// TwinCAT 3 PLC project Plc
// ProgramVersion: 3.1.4023.0
// libraries:
//   Tc2_Standard, * (Beckhoff Automation GmbH)
//   Tc2_System, * (Beckhoff Automation GmbH)
//   Tc2_Utilities, * (Beckhoff Automation GmbH)
//   Tc3_Module, * (Beckhoff Automation GmbH)
// project tree:
//   LinkedList/Master/ FB_LinkedList_Master.TcPOU, ITF_LinkedList_Master.TcIO
//   LinkedList/Node/ FB_LinkedList_Node.TcPOU, ITF_LinkedList_Node.TcIO
//   / PlcTask.TcTTO
//   POUs/Cars/ FB_Car.TcPOU, FB_CarGroup.TcPOU, ITF_Car.TcIO
//   POUs/ MAIN.TcPOU, PERFORMANCE.TcPOU
// real-time tasks:
//   TASK PlcTask: cycle T#10ms, priority 20, ADS port 350

CONFIGURATION Plc
    RESOURCE PLC ON TwinCAT3
        TASK PlcTask(INTERVAL := T#10ms, PRIORITY := 20);
        PROGRAM MAIN WITH PlcTask : MAIN;
        PROGRAM PERFORMANCE WITH PlcTask : PERFORMANCE;
    END_RESOURCE
END_CONFIGURATION

// ---- LinkedList/Master/ITF_LinkedList_Master.TcIO
INTERFACE ITF_LinkedList_Master EXTENDS ITF_LinkedList_Node

METHOD mListAdd : BOOL
VAR_INPUT
	itfNode:	ITF_LinkedList_Node;
END_VAR
END_METHOD

METHOD mListRemove : BOOL
VAR_INPUT
	itfNode:	ITF_LinkedList_Node;
END_VAR
END_METHOD

END_INTERFACE

// ---- LinkedList/Node/ITF_LinkedList_Node.TcIO
INTERFACE ITF_LinkedList_Node EXTENDS __SYSTEM.IQueryInterface

PROPERTY p_IsLinkMaster : BOOL
GET
END_GET
END_PROPERTY

PROPERTY p_ListNext : ITF_LinkedList_Node
GET
END_GET
SET
END_SET
END_PROPERTY

PROPERTY p_ListPrevious : ITF_LinkedList_Node
GET
END_GET
SET
END_SET
END_PROPERTY

END_INTERFACE

// ---- POUs/Cars/ITF_Car.TcIO
INTERFACE ITF_Car

PROPERTY p_Locked : BOOL
GET
END_GET
SET
END_SET
END_PROPERTY

END_INTERFACE

// ---- POUs/MAIN.TcPOU
PROGRAM MAIN
VAR
	fbCarFleet:		FB_CarGroup;
	fbCar_Red:		FB_Car;
	fbCar_Green:	FB_Car;
	fbCar_Blue:		FB_Car;

	fbGarage:		FB_CarGroup;
	fbCorvette:		FB_Car := ( p_LinkMaster := fbGarage );
	fbMustang:		FB_Car := ( p_LinkMaster := fbGarage );

	//Triggers
	xSellCar:		BOOL;
	xBuyCar:		BOOL;
END_VAR

VAR_TEMP
	{attribute 'hide'} 
	pCar:			POINTER TO FB_Car;
END_VAR


IF xSellCar THEN
	xSellCar := FALSE; //Reset trigger
	//Get last car in the garage list and sell it to the fleet
	IF __QUERYPOINTER(fbGarage.mListGetNode( fbGarage.ListLength - 1), pCar) THEN
		pCar^.p_LinkMaster := fbCarFleet;
	END_IF
END_IF

IF xBuyCar THEN
	xBuyCar := FALSE; //Reset trigger
	//Get first car from the fleed and add it to the garage
	IF __QUERYPOINTER(fbCarFleet.mListGetNode(0), pCar) THEN
		pCar^.p_LinkMaster := fbGarage;
	END_IF
END_IF

END_PROGRAM

// ---- POUs/Cars/FB_CarGroup.TcPOU
FUNCTION_BLOCK FB_CarGroup EXTENDS FB_LinkedList_Master IMPLEMENTS ITF_Car
VAR_INPUT
END_VAR
VAR_OUTPUT
END_VAR
VAR
END_VAR

{attribute 'monitoring' := 'call'}
PROPERTY p_Locked : BOOL
GET
VAR
	i:		UINT;
	itfCar:	ITF_Car;
END_VAR
p_Locked := TRUE;

FOR i := 0 TO ListLength DO
	IF __QUERYINTERFACE( mListGetNode(i), itfCar) THEN
		p_Locked R= NOT itfCar.p_Locked;
	END_IF
END_FOR
END_GET
SET
VAR
	i:		UINT;
	itfCar:	ITF_Car;
END_VAR
FOR i := 0 TO ListLength DO
	IF __QUERYINTERFACE( mListGetNode(i), itfCar) THEN
		itfCar.p_Locked := p_Locked;
	END_IF
END_FOR
END_SET
END_PROPERTY

END_FUNCTION_BLOCK

// ---- LinkedList/Master/FB_LinkedList_Master.TcPOU
{attribute 'hide_all_locals'}
FUNCTION_BLOCK FB_LinkedList_Master IMPLEMENTS ITF_LinkedList_Master

VAR_OUTPUT
	ListLength:		UINT;	//Length of the linked list
END_VAR

VAR
	itfHead:	ITF_LinkedList_Node;
	itfTail:	ITF_LinkedList_Node;
	
	{attribute 'no_copy'}
	it:			UINT; 					//Local iterator
	{attribute 'no_copy'}
	itfIt:		ITF_LinkedList_Node;	//Iterated node
END_VAR

METHOD mListAdd : BOOL
VAR_INPUT
	itfNode:	ITF_LinkedList_Node;
END_VAR
IF itfNode <> 0 THEN
	IF ListLength = 0 THEN
		//--Empty list--
		itfHead 				:= itfNode;
		itfTail 				:= itfNode;
		itfNode.p_ListPrevious 	:= THIS^;
		itfNode.p_ListNext		:= THIS^;
	ELSE
		//--Existing list--
		itfTail.p_ListNext 		:= itfNode;
		itfNode.p_ListNext		:= THIS^;
		itfNode.p_ListPrevious	:= itfTail;
		itfTail					:= itfNode;
	END_IF
	
	ListLength := ListLength + 1;
END_IF
END_METHOD

METHOD mListGetNode : ITF_LinkedList_Node
VAR_INPUT
	i:		UINT; //0 => Length - 1
END_VAR
//Reread/init
IF it = 0 THEN
	itfIt  	:= itfHead;
END_IF

//Reset to head
IF i = 0 THEN
	itfIt 	:= itfHead;
	it		:= 0;	
END_IF

WHILE it < i AND_THEN itfIt <> 0 AND_THEN NOT itfIt.p_IsLinkMaster  DO
	itfIt	:= itfIt.p_ListNext;
	it		:= it + 1; 
END_WHILE

WHILE it > i AND_THEN itfIt <> 0 AND_THEN NOT itfIt.p_IsLinkMaster DO
	itfIt	:= itfIt.p_ListPrevious;
	it		:= it - 1;
END_WHILE

IF itfIt <> 0 AND_THEN NOT itfIt.p_IsLinkMaster THEN
	//Node found, return interface
	mListGetNode := itfIt;
ELSE
	//Something went wrong, reset to head
	itfIt 	:= itfHead;
	it		:= 0;
END_IF
END_METHOD

METHOD mListRemove : BOOL
VAR_INPUT
	itfNode:	ITF_LinkedList_Node;
END_VAR
//Improve: Check if node is indeed in the list of this master

IF itfNode <> 0 THEN
	
	IF itfNode.p_ListPrevious <> 0 THEN
		
		IF itfNode.p_ListNext <> 0 THEN
			itfNode.p_ListPrevious.p_ListNext := itfNode.p_ListNext;
			itfNode.p_ListNext.p_ListPrevious := itfNode.p_ListPrevious;
		ELSE
			itfNode.p_ListPrevious.p_ListNext := 0;
		END_IF
		
		mListRemove := TRUE;
	END_IF

	itfNode.p_ListNext 		:= 0;
	itfNode.p_ListPrevious	:= 0;
END_IF

IF mListRemove THEN
	ListLength := MAX(0,ListLength - 1);
	
	//Reset iterator to beginning we don't know where the nodes is removed and recounting is needed
	it		:= 0;
	itfIt	:= itfHead;
END_IF
END_METHOD

PROPERTY p_IsLinkMaster : BOOL
GET
p_IsLinkMaster := TRUE;
END_GET
END_PROPERTY

PROPERTY p_ListNext : ITF_LinkedList_Node
GET
p_ListNext := itfHead;
END_GET
SET
itfHead := p_ListNext;
END_SET
END_PROPERTY

PROPERTY p_ListPrevious : ITF_LinkedList_Node
GET
p_ListPrevious := itfTail;
END_GET
SET
itfTail := p_ListPrevious;
END_SET
END_PROPERTY

END_FUNCTION_BLOCK

// ---- POUs/Cars/FB_Car.TcPOU
{attribute 'hide_all_locals'}
FUNCTION_BLOCK FB_Car EXTENDS FB_LinkedList_Node IMPLEMENTS ITF_Car

VAR
	Locked:		BOOL;
END_VAR

METHOD FB_init : BOOL
VAR_INPUT
	bInitRetains : 	BOOL; // if TRUE, the retain variables are initialized (warm start / cold start)
	bInCopyCode : 	BOOL;  // if TRUE, the instance afterwards gets moved into the copy code (online change)
END_VAR
p_LinkMaster := MAIN.fbCarFleet;
END_METHOD

{attribute 'monitoring' := 'call'}
PROPERTY p_Locked : BOOL
GET
p_Locked := Locked;
END_GET
SET
Locked := p_Locked;
END_SET
END_PROPERTY

END_FUNCTION_BLOCK

// ---- LinkedList/Node/FB_LinkedList_Node.TcPOU
{attribute 'hide_all_locals'}
FUNCTION_BLOCK FB_LinkedList_Node IMPLEMENTS ITF_LinkedList_Node

VAR
	itf_ListNext:		ITF_LinkedList_Node;
	itf_ListPrevious:	ITF_LinkedList_Node;
	itf_LinkMaster:		ITF_LinkedList_Master;
	
	{attribute 'no_copy'}
	_bInCopyCode : 		BOOL;
END_VAR

METHOD FB_exit : BOOL
VAR_INPUT
	bInCopyCode : BOOL; // if TRUE, the exit method is called for exiting an instance that is copied afterwards (online change).
END_VAR
IF NOT bInCopyCode THEN
	//Destroy and remove from list
	IF itf_LinkMaster <> 0 THEN
		itf_LinkMaster.mListRemove( THIS^ );
	END_IF
END_IF
END_METHOD

METHOD FB_init : BOOL
VAR_INPUT
	bInitRetains : 	BOOL; // if TRUE, the retain variables are initialized (warm start / cold start)
	bInCopyCode : 	BOOL;  // if TRUE, the instance afterwards gets moved into the copy code (online change)
END_VAR
_bInCopyCode 	:= bInCopyCode;
END_METHOD

METHOD FB_reinit : BOOL
VAR_INPUT
END_VAR
_bInCopyCode := FALSE; //Next set of p_LinkMaster wont be from initializing new instance during copy
END_METHOD

PROPERTY p_IsLinkMaster : BOOL
GET
p_IsLinkMaster := FALSE;
END_GET
END_PROPERTY

PROPERTY p_LinkMaster : ITF_LinkedList_Master
GET
p_LinkMaster := itf_LinkMaster;
END_GET
SET
IF NOT _bInCopyCode THEN //Set not called during process of copying function block
	
	IF itf_LinkMaster <> 0 THEN
		//Remove from old master
		itf_LinkMaster.mListRemove( THIS^ );
	END_IF

	IF p_LinkMaster <> 0 THEN
		//Add to new master
		p_LinkMaster.mListAdd( THIS^ );
		//Store master
		itf_LinkMaster := p_LinkMaster;
	END_IF

END_IF
END_SET
END_PROPERTY

PROPERTY p_ListNext : ITF_LinkedList_Node
GET
p_ListNext := itf_ListNext;
END_GET
SET
itf_ListNext := p_ListNext;
END_SET
END_PROPERTY

PROPERTY p_ListPrevious : ITF_LinkedList_Node
GET
p_ListPrevious := itf_ListPrevious;
END_GET
SET
itf_ListPrevious := p_ListPrevious;
END_SET
END_PROPERTY

END_FUNCTION_BLOCK

// ---- POUs/PERFORMANCE.TcPOU
PROGRAM PERFORMANCE
VAR CONSTANT
	iSize:			INT := 10000;
END_VAR

VAR
	fbMaster:		FB_CarGroup;
	fbCars:			ARRAY[0..iSize-1] OF FB_Car := [ iSize(( p_LinkMaster := fbMaster )) ];
	i:				INT;
	itfCar:			ITF_Car;
	
	Profiler_List: 	PROFILER;
	Profiler_Array:	PROFILER;
END_VAR

MAX_AVERAGE_MEASURES := 100;

//-----Linked list iteration----
Profiler_List( START := TRUE );
FOR i := 0 TO iSize - 1 DO
	IF __QUERYINTERFACE( fbMaster.mListGetNode( i ), itfCar) THEN
		itfCar.p_Locked := TRUE;
	END_IF
END_FOR
Profiler_List( START := FALSE );

//-----Array iteration----
Profiler_Array( START := TRUE );
FOR i := 0 TO iSize - 1 DO
	fbCars[i].p_Locked := TRUE;
END_FOR
Profiler_Array( START := FALSE );

FOR i := 0 TO iSize - 1 DO
	fbCars[i].p_Locked := NOT fbCars[i].p_Locked;
END_FOR

END_PROGRAM
